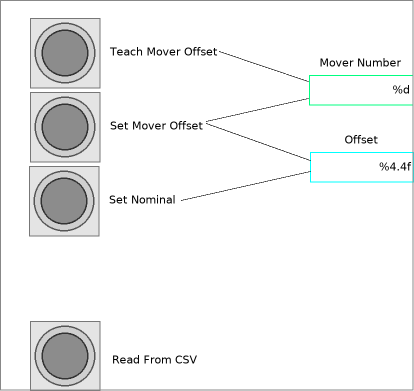
VISUALIZATION Offsets  // 414x391
    PushSwitchLed (30,18 70x70), variable: MAIN.MoverOffsets.bTeachMoverOffset, behaviour: TAP, style: Switch-PushSwitchLed-Gray
    Label (107,37 132x30), "Teach Mover Offset"
    Label (107,111 132x30), "Set Mover Offset"
    PushSwitchLed (30,92 70x70), variable: MAIN.MoverOffsets.bSetMoverOffset, behaviour: TAP, style: Switch-PushSwitchLed-Gray
    Label (106,185 115x30), "Set Nominal"
    PushSwitchLed (29,166 70x70), variable: MAIN.MoverOffsets.bSetNominal, behaviour: TAP, style: Switch-PushSwitchLed-Gray
    Textfield (309,75 104x30), "%d", text variable: MAIN.MoverOffsets.nMoverNumber
        OnMouseClick: write the text variable via VisuDialogs.Numpad, min 1, max MAIN.XTS.NumMovers, format %f.0
    Label (312,54 97x18), "Mover Number"
    Textfield (310,152 104x30), "%4.4f", text variable: MAIN.MoverOffsets.fOffset
        OnMouseClick: write the text variable via VisuDialogs.Numpad, min -100, max 100, format %f.4
    Label (313,131 97x18), "Offset"
    Label (109,345 105x30), "Read From CSV"
    PushSwitchLed (30,321 70x70), variable: MAIN.MoverOffsets.bReadCSVOffsets, behaviour: TAP, style: Switch-PushSwitchLed-Gray
    Line (219,51) (308,81)
    Line (206,121) (308,98)
    Line (206,123) (310,160)
    Line (181,200) (310,171)
END_VISUALIZATION

(* stored: Version 1.1.0.1, ProductVersion 3.1.4026.12
   Visu Offsets: Id {23829244-05ce-4b04-b7fa-3525bbd3adf7} *)
